TYPE E_CommandExecutionState : (
    COMMAND_IDLE := 0,
    COMMAND_ACCEPTED := 10,
    COMMAND_EXECUTING := 20,
    COMMAND_COMPLETED := 30,
    COMMAND_REJECTED := 40,
    COMMAND_FAILED := 50,
    COMMAND_CANCELLED := 60
); END_TYPE

(* stored: Version 1.1.0.1
   DUT E_CommandExecutionState: Id {E3000000-0000-4000-8000-000000000021} *)
